	fbSetExtendedFadeTime.ipDALICommunication := ipDALICommunication;
	fbSetFadeRate.ipDALICommunication := ipDALICommunication;
	fbSetFadeTime.ipDALICommunication := ipDALICommunication;
{endregion}
5:
{region "Start Qiescent Mode"}
	fb103StartQuiescentMode(bStart := TRUE,
							eAddressType := Tc3_DALI.E_DALIAddressType.Broadcast,
							eCommandPriority := Tc3_DALI.E_DALICommandPriority.Middle);
	IF (NOT fb103StartQuiescentMode.bBusy) THEN
		fb103StartQuiescentMode(bStart:= FALSE);
		nStep := 10;
	END_IF
{endregion}
10:
{region "Query Fade Time and Fade Rate"}
	fbQueryFadeTimeFadeRate(bStart := TRUE,
							nAddress := nAddress,
							eAddressType := eAddressType,
							eCommandPriority := E_DALICommandPriority.Middle,
							eFadeTime => eFadeTime,
							eFadeRate => eFadeRate);
	IF (NOT fbQueryFadeTimeFadeRate.bBusy) THEN
		fbQueryFadeTimeFadeRate(bStart := FALSE);
		IF (eFadeTime = 0) THEN 
			bNoFadeTime := FALSE; // Check whether Fade Time is available
			nStep := 20;
		ELSE 	 
			bNoFadeTime := TRUE;
			nStep := 0;
		END_IF
	END_IF
{endregion}
20:
{region "Query Extended Fade Time"}
	fbQueryExtendedFadeTime(bStart := TRUE,
							nAddress := nAddress,
							eAddressType := eAddressType,
							eCommandPriority := E_DALICommandPriority.Middle,
							eExtendedFadeTimeBase => eExtendedFadeTimeBase,
							eExtendedFadeTimeMultiplier => eExtendedFadeTimeMultiplier);
	IF (NOT fbQueryExtendedFadeTime.bBusy) THEN
		fbQueryExtendedFadeTime(bStart := FALSE);
		nStep := 25;
		IF (eExtendedFadeTimeMultiplier = E_DALIExtendedFadeTimeMultiplier.Disabled) THEN
			eExtendedFadeTime := E_DALIExtendedFadeTime.NoFade;
		END_IF
		IF (eExtendedFadeTimeMultiplier = E_DALIExtendedFadeTimeMultiplier.Multiplier100ms) THEN
			CASE eExtendedFadeTimeBase OF
				E_DALIExtendedFadeTimeBase.Base01:	eExtendedFadeTime := E_DALIExtendedFadeTime.onehundred;
				E_DALIExtendedFadeTimeBase.Base02:	eExtendedFadeTime := E_DALIExtendedFadeTime.twohundred;
				E_DALIExtendedFadeTimeBase.Base03:	eExtendedFadeTime := E_DALIExtendedFadeTime.threehundred;
				E_DALIExtendedFadeTimeBase.Base04:	eExtendedFadeTime := E_DALIExtendedFadeTime.fourhundred;
				E_DALIExtendedFadeTimeBase.Base05:	eExtendedFadeTime := E_DALIExtendedFadeTime.fivehundred;
				E_DALIExtendedFadeTimeBase.Base06:	eExtendedFadeTime := E_DALIExtendedFadeTime.sixhundred;
				E_DALIExtendedFadeTimeBase.Base07:	eExtendedFadeTime := E_DALIExtendedFadeTime.sevenhundred;
				E_DALIExtendedFadeTimeBase.Base08:	eExtendedFadeTime := E_DALIExtendedFadeTime.eighthundred;
				E_DALIExtendedFadeTimeBase.Base09:	eExtendedFadeTime := E_DALIExtendedFadeTime.ninehundred;
				E_DALIExtendedFadeTimeBase.Base10:	eExtendedFadeTime := E_DALIExtendedFadeTime.onethousand;
				E_DALIExtendedFadeTimeBase.Base11:	eExtendedFadeTime := E_DALIExtendedFadeTime.onethousandonehundred;
				E_DALIExtendedFadeTimeBase.Base12:	eExtendedFadeTime := E_DALIExtendedFadeTime.onethousandtwohundred;
				E_DALIExtendedFadeTimeBase.Base13:	eExtendedFadeTime := E_DALIExtendedFadeTime.onethousandthreehundred;
				E_DALIExtendedFadeTimeBase.Base14:	eExtendedFadeTime := E_DALIExtendedFadeTime.onethousandfourhundred;
				E_DALIExtendedFadeTimeBase.Base15:	eExtendedFadeTime := E_DALIExtendedFadeTime.onethousandfivehundred;
				E_DALIExtendedFadeTimeBase.Base16:	eExtendedFadeTime := E_DALIExtendedFadeTime.onethousandsixhundred;
			END_CASE
		END_IF
	 	IF (eExtendedFadeTimeMultiplier = E_DALIExtendedFadeTimeMultiplier.Multiplier1s) THEN
			CASE eExtendedFadeTimeBase OF
				E_DALIExtendedFadeTimeBase.Base01:	eExtendedFadeTime := E_DALIExtendedFadeTime.onesecond;
				E_DALIExtendedFadeTimeBase.Base02:	eExtendedFadeTime := E_DALIExtendedFadeTime.twoseconds;
				E_DALIExtendedFadeTimeBase.Base03:	eExtendedFadeTime := E_DALIExtendedFadeTime.threeseconds;
				E_DALIExtendedFadeTimeBase.Base04:	eExtendedFadeTime := E_DALIExtendedFadeTime.fourseconds;
				E_DALIExtendedFadeTimeBase.Base05:	eExtendedFadeTime := E_DALIExtendedFadeTime.fiveseconds;
				E_DALIExtendedFadeTimeBase.Base06:	eExtendedFadeTime := E_DALIExtendedFadeTime.sixseconds;
				E_DALIExtendedFadeTimeBase.Base07:	eExtendedFadeTime := E_DALIExtendedFadeTime.sevenseconds;
				E_DALIExtendedFadeTimeBase.Base08:	eExtendedFadeTime := E_DALIExtendedFadeTime.eightseconds;
				E_DALIExtendedFadeTimeBase.Base09:	eExtendedFadeTime := E_DALIExtendedFadeTime.nineseconds;
				E_DALIExtendedFadeTimeBase.Base10:	eExtendedFadeTime := E_DALIExtendedFadeTime.tenseconds;
				E_DALIExtendedFadeTimeBase.Base11:	eExtendedFadeTime := E_DALIExtendedFadeTime.elevenseconds;
				E_DALIExtendedFadeTimeBase.Base12:	eExtendedFadeTime := E_DALIExtendedFadeTime.twelveseconds;
				E_DALIExtendedFadeTimeBase.Base13:	eExtendedFadeTime := E_DALIExtendedFadeTime.thirteenseconds;
				E_DALIExtendedFadeTimeBase.Base14:	eExtendedFadeTime := E_DALIExtendedFadeTime.fourteenseconds;
				E_DALIExtendedFadeTimeBase.Base15:	eExtendedFadeTime := E_DALIExtendedFadeTime.fifteenseconds;
				E_DALIExtendedFadeTimeBase.Base16:	eExtendedFadeTime := E_DALIExtendedFadeTime.sixteenseconds;
			END_CASE
		END_IF
		IF (eExtendedFadeTimeMultiplier = E_DALIExtendedFadeTimeMultiplier.Multiplier10s) THEN
			CASE eExtendedFadeTimeBase OF
				E_DALIExtendedFadeTimeBase.Base01:	eExtendedFadeTime := E_DALIExtendedFadeTime.ten1seconds;
				E_DALIExtendedFadeTimeBase.Base02:	eExtendedFadeTime := E_DALIExtendedFadeTime.twentyseconds;
				E_DALIExtendedFadeTimeBase.Base03:	eExtendedFadeTime := E_DALIExtendedFadeTime.thirtyseconds;
				E_DALIExtendedFadeTimeBase.Base04:	eExtendedFadeTime := E_DALIExtendedFadeTime.fourtyseconds;
				E_DALIExtendedFadeTimeBase.Base05:	eExtendedFadeTime := E_DALIExtendedFadeTime.fiftyseconds;
				E_DALIExtendedFadeTimeBase.Base06:	eExtendedFadeTime := E_DALIExtendedFadeTime.sixtyseconds;
				E_DALIExtendedFadeTimeBase.Base07:	eExtendedFadeTime := E_DALIExtendedFadeTime.seventyseconds;
				E_DALIExtendedFadeTimeBase.Base08:	eExtendedFadeTime := E_DALIExtendedFadeTime.eightyseconds;
				E_DALIExtendedFadeTimeBase.Base09:	eExtendedFadeTime := E_DALIExtendedFadeTime.ninetyseconds;
				E_DALIExtendedFadeTimeBase.Base10:	eExtendedFadeTime := E_DALIExtendedFadeTime.onehundredseconds;
				E_DALIExtendedFadeTimeBase.Base11:	eExtendedFadeTime := E_DALIExtendedFadeTime.onehundredtenseconds;
				E_DALIExtendedFadeTimeBase.Base12:	eExtendedFadeTime := E_DALIExtendedFadeTime.onehundredtwentyseconds;
				E_DALIExtendedFadeTimeBase.Base13:	eExtendedFadeTime := E_DALIExtendedFadeTime.onehundredthirtyseconds;
				E_DALIExtendedFadeTimeBase.Base14:	eExtendedFadeTime := E_DALIExtendedFadeTime.onehundredfourtyseconds;
				E_DALIExtendedFadeTimeBase.Base15:	eExtendedFadeTime := E_DALIExtendedFadeTime.onehundredfiftyseconds;
				E_DALIExtendedFadeTimeBase.Base16:	eExtendedFadeTime := E_DALIExtendedFadeTime.onehundredsixtyseconds;
			END_CASE
		END_IF
		IF (eExtendedFadeTimeMultiplier = E_DALIExtendedFadeTimeMultiplier.Multiplier1min) THEN
			CASE eExtendedFadeTimeBase OF
				E_DALIExtendedFadeTimeBase.Base01:	eExtendedFadeTime := E_DALIExtendedFadeTime.oneminute;
				E_DALIExtendedFadeTimeBase.Base02:	eExtendedFadeTime := E_DALIExtendedFadeTime.twominutes;
				E_DALIExtendedFadeTimeBase.Base03:	eExtendedFadeTime := E_DALIExtendedFadeTime.threeminutes;
				E_DALIExtendedFadeTimeBase.Base04:	eExtendedFadeTime := E_DALIExtendedFadeTime.fourminutes;
				E_DALIExtendedFadeTimeBase.Base05:	eExtendedFadeTime := E_DALIExtendedFadeTime.fiveminutes;
				E_DALIExtendedFadeTimeBase.Base06:	eExtendedFadeTime := E_DALIExtendedFadeTime.sixminutes;
				E_DALIExtendedFadeTimeBase.Base07:	eExtendedFadeTime := E_DALIExtendedFadeTime.sevenminutes;
				E_DALIExtendedFadeTimeBase.Base08:	eExtendedFadeTime := E_DALIExtendedFadeTime.eightminutes;
				E_DALIExtendedFadeTimeBase.Base09:	eExtendedFadeTime := E_DALIExtendedFadeTime.nineminutes;
				E_DALIExtendedFadeTimeBase.Base10:	eExtendedFadeTime := E_DALIExtendedFadeTime.tenminutes;
				E_DALIExtendedFadeTimeBase.Base11:	eExtendedFadeTime := E_DALIExtendedFadeTime.elevenminutes;
				E_DALIExtendedFadeTimeBase.Base12:	eExtendedFadeTime := E_DALIExtendedFadeTime.twelveminutes;
				E_DALIExtendedFadeTimeBase.Base13:	eExtendedFadeTime := E_DALIExtendedFadeTime.thirteenminutes;
				E_DALIExtendedFadeTimeBase.Base14:	eExtendedFadeTime := E_DALIExtendedFadeTime.fourteenminutes;
				E_DALIExtendedFadeTimeBase.Base15:	eExtendedFadeTime := E_DALIExtendedFadeTime.fifteenminutes;
				E_DALIExtendedFadeTimeBase.Base16:	eExtendedFadeTime := E_DALIExtendedFadeTime.sixteenminutes;
			END_CASE
		END_IF
	ELSE
		eExtendedFadeTime := E_DALIExtendedFadeTime.unknown;
	END_IF
{endregion}
25:
{region "Stop Qiescent Mode"}
	fb103StopQuiescentMode(	bStart := TRUE,
							eAddressType := Tc3_DALI.E_DALIAddressType.Broadcast,
							eCommandPriority := Tc3_DALI.E_DALICommandPriority.Middle);
	IF (NOT fb103StopQuiescentMode.bBusy) THEN
		fb103StopQuiescentMode(	bStart:= FALSE);
		nStep := 0;
	END_IF
{endregion}	
1000:
{region "Set Fade Time"}
	fbSetFadeTime(	bStart := TRUE,
					nAddress := nAddress,
					eAddressType := eAddressType,
					eCommandPriority := E_DALICommandPriority.Middle,
					eFadeTime := eFadeTime);
	IF (NOT fbSetFadeTime.bBusy) THEN
		fbSetFadeTime(bStart := FALSE);
		{region " Display whether Fade Time is available²}
		IF (eFadeTime = 0) THEN
			bNoFadeTime := FALSE;
		ELSE
			bNoFadeTime := TRUE;
		END_IF
		{endregion}
		nStep := 0;
	END_IF
{endregion}
1010:
{region "Set Fade Rate"}
	fbSetFadeRate(	bStart := TRUE,
					nAddress := nAddress,
					eAddressType := eAddressType,
					eCommandPriority := E_DALICommandPriority.Middle,
					eFadeRate := eFadeRate);
	IF (NOT fbSetFadeRate.bBusy) THEN
		fbSetFadeRate(bStart := FALSE);
		nStep := 0;
	END_IF
{endregion}
1020:
{region "Set Extended Fade Time"}
	CASE eExtendedFadeTime OF
		E_DALIExtendedFadeTime.NoFade:					eExtendedFadeTimeBase := E_DALIExtendedFadeTimeBase.Unknown;
														eExtendedFadeTimeMultiplier := E_DALIExtendedFadeTimeMultiplier.Disabled;
		E_DALIExtendedFadeTime.onehundred:				eExtendedFadeTimeBase := E_DALIExtendedFadeTimeBase.Base01;
														eExtendedFadeTimeMultiplier := E_DALIExtendedFadeTimeMultiplier.Multiplier100ms;
		E_DALIExtendedFadeTime.twohundred:				eExtendedFadeTimeBase := E_DALIExtendedFadeTimeBase.Base02;
														eExtendedFadeTimeMultiplier := E_DALIExtendedFadeTimeMultiplier.Multiplier100ms;
		E_DALIExtendedFadeTime.threehundred:			eExtendedFadeTimeBase := E_DALIExtendedFadeTimeBase.Base03;
														eExtendedFadeTimeMultiplier := E_DALIExtendedFadeTimeMultiplier.Multiplier100ms;
		E_DALIExtendedFadeTime.fourhundred:				eExtendedFadeTimeBase := E_DALIExtendedFadeTimeBase.Base04;
														eExtendedFadeTimeMultiplier := E_DALIExtendedFadeTimeMultiplier.Multiplier100ms;
		E_DALIExtendedFadeTime.fivehundred:				eExtendedFadeTimeBase := E_DALIExtendedFadeTimeBase.Base05;
														eExtendedFadeTimeMultiplier := E_DALIExtendedFadeTimeMultiplier.Multiplier100ms;
		E_DALIExtendedFadeTime.sixhundred:				eExtendedFadeTimeBase := E_DALIExtendedFadeTimeBase.Base06;
														eExtendedFadeTimeMultiplier := E_DALIExtendedFadeTimeMultiplier.Multiplier100ms;
		E_DALIExtendedFadeTime.sevenhundred:			eExtendedFadeTimeBase := E_DALIExtendedFadeTimeBase.Base07;
														eExtendedFadeTimeMultiplier := E_DALIExtendedFadeTimeMultiplier.Multiplier100ms;
		E_DALIExtendedFadeTime.eighthundred:			eExtendedFadeTimeBase := E_DALIExtendedFadeTimeBase.Base08;
														eExtendedFadeTimeMultiplier := E_DALIExtendedFadeTimeMultiplier.Multiplier100ms;
		E_DALIExtendedFadeTime.ninehundred:				eExtendedFadeTimeBase := E_DALIExtendedFadeTimeBase.Base09;
														eExtendedFadeTimeMultiplier := E_DALIExtendedFadeTimeMultiplier.Multiplier100ms;
		E_DALIExtendedFadeTime.onethousand:				eExtendedFadeTimeBase := E_DALIExtendedFadeTimeBase.Base10;
														eExtendedFadeTimeMultiplier := E_DALIExtendedFadeTimeMultiplier.Multiplier100ms;
		E_DALIExtendedFadeTime.onethousandonehundred:	eExtendedFadeTimeBase := E_DALIExtendedFadeTimeBase.Base11;
														eExtendedFadeTimeMultiplier := E_DALIExtendedFadeTimeMultiplier.Multiplier100ms;
		E_DALIExtendedFadeTime.onethousandtwohundred:	eExtendedFadeTimeBase := E_DALIExtendedFadeTimeBase.Base12;
														eExtendedFadeTimeMultiplier := E_DALIExtendedFadeTimeMultiplier.Multiplier100ms;
		E_DALIExtendedFadeTime.onethousandthreehundred:	eExtendedFadeTimeBase := E_DALIExtendedFadeTimeBase.Base13;
														eExtendedFadeTimeMultiplier := E_DALIExtendedFadeTimeMultiplier.Multiplier100ms;
		E_DALIExtendedFadeTime.onethousandfourhundred:	eExtendedFadeTimeBase := E_DALIExtendedFadeTimeBase.Base14;
														eExtendedFadeTimeMultiplier := E_DALIExtendedFadeTimeMultiplier.Multiplier100ms;
		E_DALIExtendedFadeTime.onethousandfivehundred:	eExtendedFadeTimeBase := E_DALIExtendedFadeTimeBase.Base15;
														eExtendedFadeTimeMultiplier := E_DALIExtendedFadeTimeMultiplier.Multiplier100ms;
		E_DALIExtendedFadeTime.onethousandsixhundred:	eExtendedFadeTimeBase := E_DALIExtendedFadeTimeBase.Base16;
														eExtendedFadeTimeMultiplier := E_DALIExtendedFadeTimeMultiplier.Multiplier100ms;
		E_DALIExtendedFadeTime.onesecond:				eExtendedFadeTimeBase := E_DALIExtendedFadeTimeBase.Base01;
														eExtendedFadeTimeMultiplier := E_DALIExtendedFadeTimeMultiplier.Multiplier1s;
		E_DALIExtendedFadeTime.twoseconds:				eExtendedFadeTimeBase := E_DALIExtendedFadeTimeBase.Base02;
														eExtendedFadeTimeMultiplier := E_DALIExtendedFadeTimeMultiplier.Multiplier1s;
		E_DALIExtendedFadeTime.threeseconds:			eExtendedFadeTimeBase := E_DALIExtendedFadeTimeBase.Base03;
														eExtendedFadeTimeMultiplier := E_DALIExtendedFadeTimeMultiplier.Multiplier1s;
		E_DALIExtendedFadeTime.fourseconds:				eExtendedFadeTimeBase := E_DALIExtendedFadeTimeBase.Base04;
														eExtendedFadeTimeMultiplier := E_DALIExtendedFadeTimeMultiplier.Multiplier1s;
		E_DALIExtendedFadeTime.fiveseconds:				eExtendedFadeTimeBase := E_DALIExtendedFadeTimeBase.Base05;
														eExtendedFadeTimeMultiplier := E_DALIExtendedFadeTimeMultiplier.Multiplier1s;
		E_DALIExtendedFadeTime.sixseconds:				eExtendedFadeTimeBase := E_DALIExtendedFadeTimeBase.Base06;
														eExtendedFadeTimeMultiplier := E_DALIExtendedFadeTimeMultiplier.Multiplier1s;
		E_DALIExtendedFadeTime.sevenseconds:			eExtendedFadeTimeBase := E_DALIExtendedFadeTimeBase.Base07;
														eExtendedFadeTimeMultiplier := E_DALIExtendedFadeTimeMultiplier.Multiplier1s;
		E_DALIExtendedFadeTime.eightseconds:			eExtendedFadeTimeBase := E_DALIExtendedFadeTimeBase.Base08;
														eExtendedFadeTimeMultiplier := E_DALIExtendedFadeTimeMultiplier.Multiplier1s;
		E_DALIExtendedFadeTime.nineseconds:				eExtendedFadeTimeBase := E_DALIExtendedFadeTimeBase.Base09;
														eExtendedFadeTimeMultiplier := E_DALIExtendedFadeTimeMultiplier.Multiplier1s;
		E_DALIExtendedFadeTime.tenseconds:				eExtendedFadeTimeBase := E_DALIExtendedFadeTimeBase.Base10;
														eExtendedFadeTimeMultiplier := E_DALIExtendedFadeTimeMultiplier.Multiplier1s;
		E_DALIExtendedFadeTime.elevenseconds:			eExtendedFadeTimeBase := E_DALIExtendedFadeTimeBase.Base11;
														eExtendedFadeTimeMultiplier := E_DALIExtendedFadeTimeMultiplier.Multiplier1s;
		E_DALIExtendedFadeTime.twelveseconds:			eExtendedFadeTimeBase := E_DALIExtendedFadeTimeBase.Base12;
														eExtendedFadeTimeMultiplier := E_DALIExtendedFadeTimeMultiplier.Multiplier1s;
		E_DALIExtendedFadeTime.thirteenseconds:			eExtendedFadeTimeBase := E_DALIExtendedFadeTimeBase.Base13;
														eExtendedFadeTimeMultiplier := E_DALIExtendedFadeTimeMultiplier.Multiplier1s;
		E_DALIExtendedFadeTime.fourteenseconds:			eExtendedFadeTimeBase := E_DALIExtendedFadeTimeBase.Base14;
														eExtendedFadeTimeMultiplier := E_DALIExtendedFadeTimeMultiplier.Multiplier1s;
		E_DALIExtendedFadeTime.fifteenseconds:			eExtendedFadeTimeBase := E_DALIExtendedFadeTimeBase.Base15;
														eExtendedFadeTimeMultiplier := E_DALIExtendedFadeTimeMultiplier.Multiplier1s;
		E_DALIExtendedFadeTime.sixteenseconds:			eExtendedFadeTimeBase := E_DALIExtendedFadeTimeBase.Base16;
														eExtendedFadeTimeMultiplier := E_DALIExtendedFadeTimeMultiplier.Multiplier1s;
		E_DALIExtendedFadeTime.ten1seconds:				eExtendedFadeTimeBase := E_DALIExtendedFadeTimeBase.Base01;
														eExtendedFadeTimeMultiplier := E_DALIExtendedFadeTimeMultiplier.Multiplier10s;
		E_DALIExtendedFadeTime.twentyseconds:			eExtendedFadeTimeBase := E_DALIExtendedFadeTimeBase.Base02;
														eExtendedFadeTimeMultiplier := E_DALIExtendedFadeTimeMultiplier.Multiplier10s;
		E_DALIExtendedFadeTime.thirtyseconds:			eExtendedFadeTimeBase := E_DALIExtendedFadeTimeBase.Base03;
														eExtendedFadeTimeMultiplier := E_DALIExtendedFadeTimeMultiplier.Multiplier10s;
		E_DALIExtendedFadeTime.fourtyseconds:			eExtendedFadeTimeBase := E_DALIExtendedFadeTimeBase.Base04;
														eExtendedFadeTimeMultiplier := E_DALIExtendedFadeTimeMultiplier.Multiplier10s;
		E_DALIExtendedFadeTime.fiftyseconds:			eExtendedFadeTimeBase := E_DALIExtendedFadeTimeBase.Base05;
														eExtendedFadeTimeMultiplier := E_DALIExtendedFadeTimeMultiplier.Multiplier10s;
		E_DALIExtendedFadeTime.sixtyseconds:			eExtendedFadeTimeBase := E_DALIExtendedFadeTimeBase.Base06;
														eExtendedFadeTimeMultiplier := E_DALIExtendedFadeTimeMultiplier.Multiplier10s;
		E_DALIExtendedFadeTime.seventyseconds:			eExtendedFadeTimeBase := E_DALIExtendedFadeTimeBase.Base07;
														eExtendedFadeTimeMultiplier := E_DALIExtendedFadeTimeMultiplier.Multiplier10s;
		E_DALIExtendedFadeTime.eightyseconds:			eExtendedFadeTimeBase := E_DALIExtendedFadeTimeBase.Base08;
														eExtendedFadeTimeMultiplier := E_DALIExtendedFadeTimeMultiplier.Multiplier10s;
		E_DALIExtendedFadeTime.ninetyseconds:			eExtendedFadeTimeBase := E_DALIExtendedFadeTimeBase.Base09;
														eExtendedFadeTimeMultiplier := E_DALIExtendedFadeTimeMultiplier.Multiplier10s;
		E_DALIExtendedFadeTime.onehundredseconds:		eExtendedFadeTimeBase := E_DALIExtendedFadeTimeBase.Base10;
														eExtendedFadeTimeMultiplier := E_DALIExtendedFadeTimeMultiplier.Multiplier10s;
		E_DALIExtendedFadeTime.onehundredtenseconds:	eExtendedFadeTimeBase := E_DALIExtendedFadeTimeBase.Base11;
														eExtendedFadeTimeMultiplier := E_DALIExtendedFadeTimeMultiplier.Multiplier10s;
		E_DALIExtendedFadeTime.onehundredtwentyseconds:	eExtendedFadeTimeBase := E_DALIExtendedFadeTimeBase.Base12;
														eExtendedFadeTimeMultiplier := E_DALIExtendedFadeTimeMultiplier.Multiplier10s;
		E_DALIExtendedFadeTime.onehundredthirtyseconds:	eExtendedFadeTimeBase := E_DALIExtendedFadeTimeBase.Base13;
														eExtendedFadeTimeMultiplier := E_DALIExtendedFadeTimeMultiplier.Multiplier10s;
		E_DALIExtendedFadeTime.onehundredfourtyseconds:	eExtendedFadeTimeBase := E_DALIExtendedFadeTimeBase.Base14;
														eExtendedFadeTimeMultiplier := E_DALIExtendedFadeTimeMultiplier.Multiplier10s;
		E_DALIExtendedFadeTime.onehundredfiftyseconds:	eExtendedFadeTimeBase := E_DALIExtendedFadeTimeBase.Base15;
														eExtendedFadeTimeMultiplier := E_DALIExtendedFadeTimeMultiplier.Multiplier10s;
		E_DALIExtendedFadeTime.onehundredsixtyseconds:	eExtendedFadeTimeBase := E_DALIExtendedFadeTimeBase.Base16;
														eExtendedFadeTimeMultiplier := E_DALIExtendedFadeTimeMultiplier.Multiplier10s;
		E_DALIExtendedFadeTime.oneminute:				eExtendedFadeTimeBase := E_DALIExtendedFadeTimeBase.Base01;
														eExtendedFadeTimeMultiplier := E_DALIExtendedFadeTimeMultiplier.Multiplier1min;
		E_DALIExtendedFadeTime.twominutes:				eExtendedFadeTimeBase := E_DALIExtendedFadeTimeBase.Base02;
														eExtendedFadeTimeMultiplier := E_DALIExtendedFadeTimeMultiplier.Multiplier1min;
		E_DALIExtendedFadeTime.threeminutes:			eExtendedFadeTimeBase := E_DALIExtendedFadeTimeBase.Base03;
														eExtendedFadeTimeMultiplier := E_DALIExtendedFadeTimeMultiplier.Multiplier1min;
		E_DALIExtendedFadeTime.fourminutes:				eExtendedFadeTimeBase := E_DALIExtendedFadeTimeBase.Base04;
														eExtendedFadeTimeMultiplier := E_DALIExtendedFadeTimeMultiplier.Multiplier1min;
		E_DALIExtendedFadeTime.fiveminutes:				eExtendedFadeTimeBase := E_DALIExtendedFadeTimeBase.Base05;
														eExtendedFadeTimeMultiplier := E_DALIExtendedFadeTimeMultiplier.Multiplier1min;
		E_DALIExtendedFadeTime.sixminutes:				eExtendedFadeTimeBase := E_DALIExtendedFadeTimeBase.Base06;
														eExtendedFadeTimeMultiplier := E_DALIExtendedFadeTimeMultiplier.Multiplier1min;
		E_DALIExtendedFadeTime.sevenminutes:			eExtendedFadeTimeBase := E_DALIExtendedFadeTimeBase.Base07;
														eExtendedFadeTimeMultiplier := E_DALIExtendedFadeTimeMultiplier.Multiplier1min;
		E_DALIExtendedFadeTime.eightminutes:			eExtendedFadeTimeBase := E_DALIExtendedFadeTimeBase.Base08;
														eExtendedFadeTimeMultiplier := E_DALIExtendedFadeTimeMultiplier.Multiplier1min;
		E_DALIExtendedFadeTime.nineminutes:				eExtendedFadeTimeBase := E_DALIExtendedFadeTimeBase.Base09;
														eExtendedFadeTimeMultiplier := E_DALIExtendedFadeTimeMultiplier.Multiplier1min;
		E_DALIExtendedFadeTime.tenminutes:				eExtendedFadeTimeBase := E_DALIExtendedFadeTimeBase.Base10;
														eExtendedFadeTimeMultiplier := E_DALIExtendedFadeTimeMultiplier.Multiplier1min;
		E_DALIExtendedFadeTime.elevenminutes:			eExtendedFadeTimeBase := E_DALIExtendedFadeTimeBase.Base11;
														eExtendedFadeTimeMultiplier := E_DALIExtendedFadeTimeMultiplier.Multiplier1min;
		E_DALIExtendedFadeTime.twelveminutes:			eExtendedFadeTimeBase := E_DALIExtendedFadeTimeBase.Base12;
														eExtendedFadeTimeMultiplier := E_DALIExtendedFadeTimeMultiplier.Multiplier1min;
		E_DALIExtendedFadeTime.thirteenminutes:			eExtendedFadeTimeBase := E_DALIExtendedFadeTimeBase.Base13;
														eExtendedFadeTimeMultiplier := E_DALIExtendedFadeTimeMultiplier.Multiplier1min;
		E_DALIExtendedFadeTime.fourteenminutes:			eExtendedFadeTimeBase := E_DALIExtendedFadeTimeBase.Base14;
														eExtendedFadeTimeMultiplier := E_DALIExtendedFadeTimeMultiplier.Multiplier1min;
		E_DALIExtendedFadeTime.fifteenminutes:			eExtendedFadeTimeBase := E_DALIExtendedFadeTimeBase.Base15;
														eExtendedFadeTimeMultiplier := E_DALIExtendedFadeTimeMultiplier.Multiplier1min;
		E_DALIExtendedFadeTime.sixteenminutes:			eExtendedFadeTimeBase := E_DALIExtendedFadeTimeBase.Base16;
														eExtendedFadeTimeMultiplier := E_DALIExtendedFadeTimeMultiplier.Multiplier1min;
		E_DALIExtendedFadeTime.unknown:					eExtendedFadeTimeBase := E_DALIExtendedFadeTimeBase.Unknown;
														eExtendedFadeTimeMultiplier := E_DALIExtendedFadeTimeMultiplier.Unknown;
	END_CASE
	fbSetExtendedFadeTime(	bStart := TRUE,
							nAddress := nAddress,
							eAddressType := eAddressType,
							eCommandPriority := E_DALICommandPriority.Middle,
							eExtendedFadeTimeBase := eExtendedFadeTimeBase,
							eExtendedFadeTimeMultiplier := eExtendedFadeTimeMultiplier);
	IF (NOT fbSetExtendedFadeTime.bBusy) THEN
		fbSetExtendedFadeTime(bStart := FALSE);
		nStep := 0;
	END_IF
{endregion}
END_CASE

END_FUNCTION_BLOCK

// ---- POUs/DALI/DALI_Setup/FBs/FB_Part103Addressing.TcPOU
FUNCTION_BLOCK FB_Part103Addressing
VAR_INPUT
	ipDALICommunication			:	I_DALICommunication;
END_VAR
VAR_OUTPUT
	bBusy						:	BOOL;
END_VAR
VAR
	{region "Visu"}
	bScanDevices				:	BOOL;
	bStartChangeAddress			:	BOOL;
	bStartRandomAddressing		:	BOOL;
	nStartAddress				:	BYTE;
	bNewInstallation			:	BOOL;
	bOpticalFeedback			:	BOOL;
	bHideWaitSymbol				:	BOOL := TRUE;
	{endregion}
	nStep						:	INT;
	nAddress					:	INT;
	aChangeAddressList			:	ARRAY [0..63] OF ST_DALIChangeAddressList;
	aShortAddress				:	ARRAY [0..63] OF INT;
	aNoShortAddress				:	ARRAY [0..63] OF BOOL;
	nRow						:	INT;
	nHideLine					:	INT; // Variable to find out how many rows are used

	fb103StartQuiescentMode		:	FB_DALI103StartQuiescentMode(0);
	fb103StopQuiescentMode		:	FB_DALI103StopQuiescentMode(0);
	fb103Addressing				:	FB_DALI103Addressing(0);
	fb103QueryRandomAddress		:	FB_DALI103QueryRandomAddress(0);
	fb103ChangeAddresses		:	FB_DALI103ChangeAddresses(0);
END_VAR

{region "Detect Commands"}
IF (bStartRandomAddressing AND (nStep = 0)) THEN
	nStep := 5;
	bStartRandomAddressing := FALSE;
	bHideWaitSymbol := FALSE;
END_IF

IF (bScanDevices AND (nStep = 0)) THEN
	nStep := 20;
	nAddress :=0;
	bScanDevices := FALSE;
	bHideWaitSymbol := FALSE;
END_IF

IF (bStartChangeAddress AND (nStep = 0)) THEN
	nStep := 60;
	bStartChangeAddress := FALSE;
	bHideWaitSymbol := FALSE;
END_IF
{endregion}
{region "Manage Dialog Selection}
IF (nStep = 0) THEN
	bBusy := FALSE;
ELSE
	bBusy := TRUE;
END_IF
{endregion}	 
{region "Execute Commands"}
CASE nStep OF
0:
{region "Init"}
	bScanDevices := FALSE;
	bStartChangeAddress := FALSE;
	bStartRandomAddressing := FALSE;
	bHideWaitSymbol := TRUE;

	fb103StartQuiescentMode.ipDALICommunication := ipDALICommunication;
	fb103StopQuiescentMode.ipDALICommunication := ipDALICommunication;
	fb103Addressing.ipDALICommunication := ipDALICommunication;
	fb103QueryRandomAddress.ipDALICommunication := ipDALICommunication;
	fb103ChangeAddresses.ipDALICommunication := ipDALICommunication;
{endregion}
5:
{region "Start Qiescent Mode"}
	fb103StartQuiescentMode(bStart := TRUE,
							eAddressType := Tc3_DALI.E_DALIAddressType.Broadcast,
							eCommandPriority := Tc3_DALI.E_DALICommandPriority.Middle);
	IF (NOT fb103StartQuiescentMode.bBusy) THEN
		fb103StartQuiescentMode(bStart:= FALSE);
		nStep := 10;
	END_IF
{endregion}
10:
{region "RandomAddressing"}
	IF bNewInstallation THEN
		fb103Addressing.nOptions := Tc3_DALI.GVL.cCompleteNewInstallation;
	END_IF

	IF bOpticalFeedback THEN
		fb103Addressing.nOptions := Tc3_DALI.GVL.cOpticalFeedback;
	END_IF

	IF bNewInstallation AND bOpticalFeedback THEN
		fb103Addressing.nOptions := Tc3_DALI.GVL.cCompleteNewInstallation OR Tc3_DALI.GVL.cOpticalFeedback;
	END_IF
	fb103Addressing(bStart := TRUE,
					nStartWithShortAddress := nStartAddress);
	IF (NOT fb103Addressing.bBusy) THEN
		fb103Addressing(bStart := FALSE);
		nStep := 15;
	END_IF
{endregion}
15:
{region "Stop Qiescent Mode"}
	fb103StopQuiescentMode(	bStart := TRUE,
							eAddressType := Tc3_DALI.E_DALIAddressType.Broadcast,
							eCommandPriority := Tc3_DALI.E_DALICommandPriority.Middle);
	IF (NOT fb103StopQuiescentMode.bBusy) THEN
		fb103StopQuiescentMode(	bStart:= FALSE);
		nStep := 0;
	END_IF
{endregion}
{region "Read Existing Addresses"}
20:
{region "Start Qiescent Mode"}
	fb103StartQuiescentMode(bStart := TRUE,
							eAddressType := Tc3_DALI.E_DALIAddressType.Broadcast,
							eCommandPriority := Tc3_DALI.E_DALICommandPriority.Middle);
	IF (NOT fb103StartQuiescentMode.bBusy) THEN
		fb103StartQuiescentMode(bStart:= FALSE);
		nStep := 30;
	END_IF
{endregion}
30:
	// Query of the new random addresses to find out which short addresses are existing.
	fb103QueryRandomAddress (	bStart := TRUE,
								nAddress := TO_BYTE(nAddress),
								eAddressType := Tc3_DALI.E_DALIAddressType.Short,
								nRandomAddress => aChangeAddressList[nAddress].nRandomAddress);
	IF (NOT fb103QueryRandomAddress.bBusy) THEN
		fb103QueryRandomAddress(bStart := FALSE);
		nAddress := nAddress + 1;
		IF (nAddress > 63) THEN
			nStep := 40;
		END_IF
	END_IF
40:
	// Write the existing short addresses into the table 
	nRow := 0;
	FOR nAddress := 0 TO 63 DO
		IF (aChangeAddressList[nAddress].nRandomAddress > 0) THEN
			aChangeAddressList[nRow].nOldAddress := TO_BYTE(nAddress);
			nRow := nRow + 1;
		END_IF
	END_FOR
	nStep := 50;
50:
	// Hide unused rows in the table
	nHideLine := 0;
	FOR nAddress := 0 TO 63 DO 
		IF (aChangeAddressList[nAddress].nRandomAddress <> 0) THEN
			aShortAddress[nHideLine] := nAddress;
			nHideLine := nHideLine + 1;
		END_IF
	END_FOR
	FOR nAddress := nHideLine TO 63 DO 
		aNoShortAddress[nAddress] := TRUE;
	END_FOR
	FOR nAddress := 0 TO (nHideLine - 1) DO
		aNoShortAddress[nAddress] := FALSE;
	END_FOR
	aChangeAddressList[nHideLine].nOldAddress := 255;
	FOR nAddress := 0 TO nHideLine DO
		aChangeAddressList[nAddress].nNewAddress := aChangeAddressList[nAddress].nOldAddress;
	END_FOR
	nStep := 55;
{endregion}
55:
{region "Stop Qiescent Mode"}
	fb103StopQuiescentMode(	bStart := TRUE,
							eAddressType := Tc3_DALI.E_DALIAddressType.Broadcast,
							eCommandPriority := Tc3_DALI.E_DALICommandPriority.Middle);
	IF (NOT fb103StopQuiescentMode.bBusy) THEN
		fb103StopQuiescentMode(	bStart:= FALSE);
		nStep := 0;
	END_IF
{endregion}
60:
{region "Write Changed Addresses}
	fb103ChangeAddresses(	bStart := TRUE,
							aChangeAddressList := aChangeAddressList);
	IF (NOT fb103ChangeAddresses.bBusy) THEN
		fb103ChangeAddresses(	bStart := FALSE,
								aChangeAddressList := aChangeAddressList);
		nStep := 70;
	END_IF
{endregion}
70:
{region "Write New Address To Old Address}
	FOR nAddress := 0 TO 63 DO
		aChangeAddressList[nAddress].nOldAddress := aChangeAddressList[nAddress].nNewAddress;
	END_FOR
	nStep := 0;
{endregion}
END_CASE

END_FUNCTION_BLOCK

// ---- POUs/DALI/PRGs/EnergyData/P_DALI_Energy_Line.TcPOU
(*
EnergyReporting reads ActiveEnergy (part 252) for all present ballasts on all (configured) DALI-lines where GVL_DALI.g_arrEnergyData[*DALI-line*,*ballast*].bHasEnergyData is TRUE.
Results are stored in GVL_DALI.g_arrEnergyData[*DALI-line*,*ballast*].fActiveEnergy. Energy Data for individual ballasts is NOT persistent.
The engergy sum per DALI-Line (Wh) and Total Energy (kWh) are persistent.

If bCheckActiveEnergy is TRUE, all present ballasts are queried for ActiveEnergy and bHasEnergyData is updated accordingly.
This will result in errors for any ballast that does not comply with part 252.
Errors will not be triggered for activations where bCheckActiveEnergy is FALSE.

After shutdown or download to PLC EnergyReporting is activated automatically internally with bCheckActiveEnergy set to TRUE

EnergyReporting is activated automatically at TOD 0:00, 6:00, 12:00, 18:00 (configurable)

NB:	The priority of commands are set to "middle" internally. Updating all lines will take a couple of minutes to finish, so be patient.
	Other critical commands on the DALI-lines take priotity.
	Add appropriate communication immediately after configuration of a new KL6821 terminal.
	That is, arrfbDALI_EnergyReporting[*DALI-Line*].ipDALICommunication := P_DALI_Background.arrfbKL6821Communication[*DALI-Line*];
*)


PROGRAM P_DALI_Energy_Line
VAR
	arrfbDALI_EnergyReporting	: ARRAY[1..SH_Light.DALI_Param.MAX_DALIV2_LINES] OF FB_DALI_EnergyReporting;
	fbDALI_EnergyDataManagement	: SH_Light.FB_DALI_EnergyDataManagement;
	nNumOfEnergyLines			: BYTE;
	bReadEnergyDataAllLines		: BOOL;
	bReportingDone				: BOOL;
	fbRTrig_ReportingDone		: R_TRIG;
	bRTrigReportingDone			: BOOL;
	
	//Task scheduling
	stLocalSystemTime 		: TIMESTRUCT;
	fbLocalSystemTime 		: FB_LocalSystemTime;
	bGetTime 				: BOOL := TRUE;
	tTimeOut 				: TIME := DEFAULT_ADS_TIMEOUT;
	bLocalSystemTimeValid	: BOOL;
	tzID       				: E_TimeZoneID := eTimeZoneID_Invalid;
	
	tdSystemTime			: TOD;
	btestTodCompare			: BOOL;
	
	
END_VAR
VAR CONSTANT
	tdMidnight						: TOD := TOD#0:0:0;
	tdMorning						: TOD := TOD#6:0:0;
	tdMidDay						: TOD := TOD#12:0:0;
	tdEvening						: TOD := TOD#18:0:0;
	tCheckDuration					: TIME:= T#5S;
	tdTestsum						: TOD := (tdMidnight + tCheckDuration);
END_VAR

VAR PERSISTENT
	arrDaliLineEnergySumWh				: ARRAY[1..SH_Light.DALI_Param.MAX_DALIV2_LINES] OF LREAL;
	fTotalEnergyWh						: LREAL;
	nMaxControlGearOperatingHours		: UINT;
END_VAR


arrfbDALI_EnergyReporting[1].ipDALICommunication := P_DALI_Background.arrfbKL6821Communication[1];
arrfbDALI_EnergyReporting[2].ipDALICommunication := P_DALI_Background.arrfbKL6821Communication[2];
arrfbDALI_EnergyReporting[3].ipDALICommunication := P_DALI_Background.arrfbKL6821Communication[3];
//arrfbDALI_EnergyReporting[4].ipDALICommunication := P_DALI_Background.arrfbKL6821Communication[4];
//arrfbDALI_EnergyReporting[5].ipDALICommunication := P_DALI_Background.arrfbKL6821Communication[5];
//arrfbDALI_EnergyReporting[6].ipDALICommunication := P_DALI_Background.arrfbKL6821Communication[6]; // for more update SH_Light.DALI_Param.MAX_DALIV2_LINES

nNumOfEnergyLines := 3;

fbLocalSystemTime(
	sNetID:= '', 
	bEnable:= bGetTime, 
	dwCycle:= 2, // cycle time (in seconds) , Synchronization  every 2 seconds.
	dwOpt:= 1, //Bit 0: If this is set, the Windows system time is additionally synchronized cyclically with the hardware clock (RTC) (corresponds to the function NT_SetTimeToRTCTime).
	tTimeout:= tTimeOut, 
	bValid=> bLocalSystemTimeValid, 
	systemTime=> stLocalSystemTime, 
	tzID=> tzID);
	
tdSystemTime := SYSTEMTIME_TO_TOD(systemTime := stLocalSystemTime);
IF	((tdSystemTime > tdMidnight AND tdSystemTime < (tdMidnight + tCheckDuration)) OR (tdSystemTime > tdMorning AND tdSystemTime < (tdMorning + tCheckDuration)) OR
	(tdSystemTime > tdMidDay AND tdSystemTime < (tdMidDay + tCheckDuration)) OR (tdSystemTime > tdEvening AND tdSystemTime < (tdEvening + tCheckDuration))) THEN
	bReadEnergyDataAllLines := TRUE;
END_IF

fbDALI_EnergyDataManagement(
	NumOfEnergyLines				:= nNumOfEnergyLines,
	bReadEnergyDataAllLines 		:= bReadEnergyDataAllLines,
	arrfbDALI_EnergyReporting		:= arrfbDALI_EnergyReporting,
	arrDaliLineEnergySum			:= arrDaliLineEnergySumWH,
	fTotalEnergyWh					:= fTotalEnergyWh,
	nMaxControlGearOperatingHours	:= nMaxControlGearOperatingHours,
	bReportingDone					=> bReportingDone
);
GVL_AHDataModbus.nTotalEnergy10kWh := TO_UINT(TRUNC(fTotalEnergyWh*EXPT(10,-4)));  //FB_DALI_EnergyDataManagement makes sure only positive values are returned. As so, conversion from REAL to UINT is appropriate
GVL_AHDataModbus.nMaxControlGearOperatingHours := nMaxControlGearOperatingHours;

END_PROGRAM

// ---- POUs/EnOcean/P_EnOcean.TcPOU
PROGRAM P_EnOcean
VAR
	fbKL6581			: FB_KL6581;
	stKL6581_in  AT %I* : KL6581_INPUT;
	stKL6581_out AT %Q*	: KL6581_OUTPUT;
	stKL6581			: STR_KL6581;
	bInitCom			: BOOL := TRUE;
	
	arrEnOcean_Search	: ARRAY [1..8] OF FB_EnOcean_Search;
	nSearchIdx			: BYTE;
	bSerach				: BOOL;
	arrDevices			: ARRAY [1..8] OF INT;
	arrID					: ARRAY [1..8, 0..255] OF DWORD;

	//Trykknapper Atrium
	fbAtriumNiveau_Tryk_PladeB_Old				: FB_Rec_RPS_Switch;
	fbAtriumNiveau_Tryk_PladeB						: FB_Rec_RPS_Switch;
	fbAtriumNiveau_Tryk_Sevice						: FB_Rec_RPS_Switch;

	//Trykknapper på gange
	fbGang_4_413_Tryk_Pendler    						: FB_Rec_RPS_Switch;	
	
	//Trykknapper i rum
	fbRum_3_429_Tryk_Indgang							: FB_Rec_RPS_Switch;
	fbRum_3_429_Tryk_Ekstra							: FB_Rec_RPS_Switch;
	
	fbRum_4_407_Tryk_Indgang1						: FB_Rec_RPS_Switch;
	fbRum_4_407_Tryk_Indgang2						: FB_Rec_RPS_Switch;
	
	fbRum_4_411_Tryk_Indgang							: FB_Rec_RPS_Switch;
	fbRum_4_411_Tryk_Ekstra							: FB_Rec_RPS_Switch;
	
	//fbRum_1_215_Tryk											: FB_Rec_RPS_Switch;
	
END_VAR

VAR CONSTANT
	byNode_1: BYTE := 1;
	byNode_2: BYTE := 2;
	byNode_3: BYTE := 3;
	byNode_4: BYTE := 4;
	byNode_5: BYTE := 5;
	byNode_6: BYTE := 6;
	byNode_7: BYTE := 7;
	byNode_8: BYTE := 8;
END_VAR


(* Kommunikation mit der KL6581. *)
(* Communication with the KL6581. *)
fbKL6581(
	bInit			:= bInitCom,
	nIdx			:= 2,
	stKL6581_in		:= stKL6581_In,
	stKL6581_out	:= stKL6581_Out,
	bReady			=> ,
	bBusy			=> ,
	bError			=> ,
	iErrorID		=> ,
	str_KL6581		=> stKL6581);
	
GVL_AHDataModbus.EnOceanError	:= TO_UINT(fbKL6581.iErrorID);

(* Warten bis der Kommunikationsbaustein initialisiert wurde.*)
(* Wait until the communication function block has been initialized. *)
IF (NOT fbKL6581.bReady) THEN
	RETURN;
END_IF

FOR nSearchIdx:= 1 TO 8 DO
	arrEnOcean_Search[nSearchIdx](
		bStart:= TRUE, 
		str_KL6581:= stKL6581 , 
		byNode:= nSearchIdx, 
		bReceive=> , 
		iDevices=>arrDevices[nSearchIdx] , 
		ar_ID=> );
		
		MEMCPY(ADR(arrID[nSearchIdx,0]), ADR(arrEnOcean_Search[nSearchIdx].ar_ID), SIZEOF(arrEnOcean_Search[nSearchIdx].ar_ID)); 
END_FOR

//Atrium
A_AtriumNiveau();

//Gange
A_Gang_4_413();

//Rum
A_Rum_3_429();
A_Rum_4_407();
A_Rum_4_411();

ACTION A_AtriumNiveau:
fbAtriumNiveau_Tryk_PladeB_Old(
	str_KL6581:=stKL6581 , 
	byNode:=0, 
	dw_ID:= 16#0029EE85, 
	str_EnOceanSwitch=> GVL_EnOcean.strEnOceanSwitch_AtriumNiveau_PladeB_Old,
	by_Node=> , 
	bReceive=> );
	
	fbAtriumNiveau_Tryk_PladeB(
	str_KL6581:=stKL6581 , 
	byNode:=0, 
	dw_ID:= 16#0029B92D, 
	str_EnOceanSwitch=> GVL_EnOcean.strEnOceanSwitch_AtriumNiveau_PladeB,
	by_Node=> , 
	bReceive=> );
	
(*
fbAtriumNiveau_Tryk_Sevice(
	str_KL6581:=stKL6581 , 
	byNode:=0, 
	dw_ID:= 16#00FEE4FE87, 
	str_EnOceanSwitch=> GVL_EnOcean.strEnOceanSwitch_AtriumNiveau_Service, 
	by_Node=> , 
	bReceive=> );
*)
END_ACTION

ACTION A_Gang_4_413:
fbGang_4_413_Tryk_Pendler(
	str_KL6581:=stKL6581 , 
	byNode:=byNode_2, 
	dw_ID:= 16#0029AAC6, 
	str_EnOceanSwitch=> GVL_EnOcean.strEnOceanSwitch_Gang_4_413_Pendler, 
	by_Node=> , 
	bReceive=> );
END_ACTION

ACTION A_Rum_3_429:
fbRum_3_429_Tryk_Indgang(
	str_KL6581:=stKL6581 , 
	byNode:=byNode_2, 
	dw_ID:= 16#0029AD76, 
	str_EnOceanSwitch=> GVL_EnOcean.strEnOceanSwitch_Rum_3_429_Indgang, 
	by_Node=> , 
	bReceive=> );
	
	fbRum_3_429_Tryk_Ekstra(
	str_KL6581:=stKL6581 , 
	byNode:=byNode_2, 
	dw_ID:= 16#0029ABAC, 
	str_EnOceanSwitch=> GVL_EnOcean.strEnOceanSwitch_Rum_3_429_Ekstra, 
	by_Node=> , 
	bReceive=> );
END_ACTION

ACTION A_Rum_4_407:
fbRum_4_407_Tryk_Indgang1(
	str_KL6581:=stKL6581 , 
	byNode:=byNode_2, 
	dw_ID:= 16#0, 
	str_EnOceanSwitch=> GVL_EnOcean.strEnOceanSwitch_Rum_4_407_Indgang1, 
	by_Node=> , 
	bReceive=> );
	
	fbRum_4_407_Tryk_Indgang2(
	str_KL6581:=stKL6581 , 
	byNode:=byNode_2, 
	dw_ID:= 16#0, 
	str_EnOceanSwitch=> GVL_EnOcean.strEnOceanSwitch_Rum_4_407_Indgang2, 
	by_Node=> , 
	bReceive=> );
END_ACTION

ACTION A_Rum_4_411:
fbRum_4_411_Tryk_Indgang(
	str_KL6581:=stKL6581 , 
	byNode:=byNode_2, 
	dw_ID:= 16#0029ABB2, 
	str_EnOceanSwitch=> GVL_EnOcean.strEnOceanSwitch_Rum_4_411_Indgang, 
	by_Node=> , 
	bReceive=> );
	
	fbRum_4_411_Tryk_Ekstra(
	str_KL6581:=stKL6581 , 
	byNode:=byNode_2, 
	dw_ID:= 16#0029AADD, 
	str_EnOceanSwitch=> GVL_EnOcean.strEnOceanSwitch_Rum_4_411_Ekstra, 
	by_Node=> , 
	bReceive=> );
END_ACTION

END_PROGRAM

// ---- POUs/MAIN.TcPOU
PROGRAM MAIN
VAR
	nAlive: INT;
	breset: BOOL;
	nDemoVariable : INT;
	nCX8200_State	AT %I*	: UINT;
END_VAR

VAR PERSISTENT
	nDemoVar_Persist: INT;
END_VAR

nAlive:= nAlive + 1;
GVL_AHDataModbus.nCX8200_State_MB := nCX8200_State;

//Håndterer vedvarende data
	P_SystemDK.M_nCyclic(bReset := breset );
//Håndterer DALI-diagnostik (run once)
	P_DALI_DIAG();
//Håndterer adressering		
	DALI_Commissioning();
//Håndterer energirapportering
	P_DALI_Energy_Line();
//Håndterer moodbus-kommunikation (kun PLC-oversigt)
	P_AHModbusComm();

//Håndterer individuel lyskontrol i lokaler
	//Gange
	P_Gang_3_409();
	P_Gang_4_410A();
	P_Gang_4_413();

	
	//Rum
	P_Rum_3_429();
	P_Rum_4_407();
	P_Rum_4_411();
	
//Testprogrammer
	//P_DALI_Energy_Firmware_Test();

END_PROGRAM

// ---- POUs/Alle_Rum/Gange/Gang_3_409/Visualization_4_308_1.TcVIS
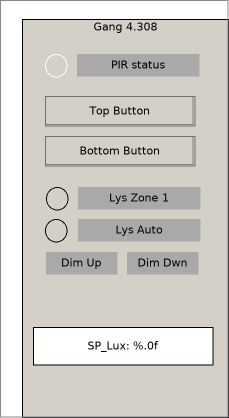
VISUALIZATION Visualization_4_308_1  // 229x418
    RoundedRectangle (22,19 207x399), "Gang 4.308"
    Rectangle (33,327 180x38), "SP_Lux: %.0f", text variable: P_Gang_4_308.arrfbLysGruppe[1].fbLightCtrl.fLuxZone1
    Button (45,96 150x30), "Top Button"
        tap P_Gang_4_308.bButtonZone1_Visu
    Button (45,136 150x30), "Bottom Button"
        tap P_Gang_4_308.bBottomButtonZone1_Visu
    Ellipse (46,187 22x23), colour toggle: P_Gang_4_308.fbLys.fbLightCtrl.bOnZone1
    Rectangle (78,187 122x22), "Lys Zone 1"
    Rectangle (46,252 71x22), "Dim Up", colour toggle: P_Gang_4_308.arrfbLysGruppe[1].fbLightCtrl.bDimUp
    Rectangle (127,252 71x22), "Dim Dwn", colour toggle: P_Gang_4_308.arrfbLysGruppe[1].fbLightCtrl.bDimDwn
    Ellipse (45,219 22x23), colour toggle: P_Gang_4_308.arrfbLysGruppe[1].fbLightCtrl.bAutoZone1
    Rectangle (78,219 122x22), "Lys Auto"
    Ellipse (45,54 22x23), colour toggle: P_Gang_4_308.arrfbLysGruppe[1].fbLightCtrl.bPIR
    Rectangle (77,54 122x22), "PIR status"
END_VISUALIZATION

// ---- POUs/Alle_Rum/Gange/Gang_4_313/Visualization_4_308_1_1.TcVIS
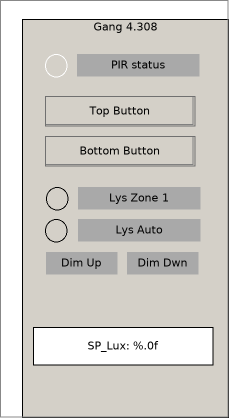
VISUALIZATION Visualization_4_308_1_1  // 229x418
    RoundedRectangle (22,19 207x399), "Gang 4.308"
    Rectangle (33,327 180x38), "SP_Lux: %.0f", text variable: P_Gang_4_308.arrfbLysGruppe[1].fbLightCtrl.fLuxZone1
    Button (45,96 150x30), "Top Button"
        tap P_Gang_4_308.bButtonZone1_Visu
    Button (45,136 150x30), "Bottom Button"
        tap P_Gang_4_308.bBottomButtonZone1_Visu
    Ellipse (46,187 22x23), colour toggle: P_Gang_4_308.fbLys.fbLightCtrl.bOnZone1
    Rectangle (78,187 122x22), "Lys Zone 1"
    Rectangle (46,252 71x22), "Dim Up", colour toggle: P_Gang_4_308.arrfbLysGruppe[1].fbLightCtrl.bDimUp
    Rectangle (127,252 71x22), "Dim Dwn", colour toggle: P_Gang_4_308.arrfbLysGruppe[1].fbLightCtrl.bDimDwn
    Ellipse (45,219 22x23), colour toggle: P_Gang_4_308.arrfbLysGruppe[1].fbLightCtrl.bAutoZone1
    Rectangle (78,219 122x22), "Lys Auto"
    Ellipse (45,54 22x23), colour toggle: P_Gang_4_308.arrfbLysGruppe[1].fbLightCtrl.bPIR
    Rectangle (77,54 122x22), "PIR status"
END_VISUALIZATION

// ---- POUs/Alle_Rum/Rum_Med_DALI_Pir/Rum_4_411/Visualization_5_356_2_1_1_3_2.TcVIS
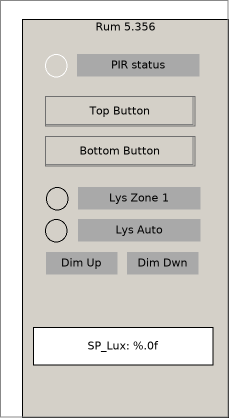
VISUALIZATION Visualization_5_356_2_1_1_3_2  // 229x418
    RoundedRectangle (22,19 207x399), "Rum 5.356"
    Rectangle (33,327 180x38), "SP_Lux: %.0f", text variable: P_Rum_5_356.arrfbLysGruppe[1].fbLightCtrl.fLuxZone1
    Button (45,96 150x30), "Top Button"
        tap P_Rum_5_356.bTopButtonZone1_Visu
    Button (45,136 150x30), "Bottom Button"
        tap P_Rum_5_356.bBottomButtonZone1_Visu
    Ellipse (46,187 22x23), colour toggle: P_Rum_5_356.arrfbLysGruppe[1].fbLightCtrl.bOnZone1
    Rectangle (78,187 122x22), "Lys Zone 1"
    Rectangle (46,252 71x22), "Dim Up", colour toggle: P_Rum_5_356.arrfbLysGruppe[1].fbLightCtrl.bDimUp
    Rectangle (127,252 71x22), "Dim Dwn", colour toggle: P_Rum_5_356.arrfbLysGruppe[1].fbLightCtrl.bDimDwn
    Ellipse (45,219 22x23), colour toggle: P_Rum_5_356.arrfbLysGruppe[1].fbLightCtrl.bAutoZone1
    Rectangle (78,219 122x22), "Lys Auto"
    Ellipse (45,54 22x23), colour toggle: P_Gang_5_356.arrfbLysGruppe[1].fbLightCtrl.bPIR
    Rectangle (77,54 122x22), "PIR status"
END_VISUALIZATION

// ---- POUs/Alle_Rum/Rum_Med_DALI_Pir/Rum_4_407/Visualization_5_356_2_1_1_6_1_6_1.TcVIS
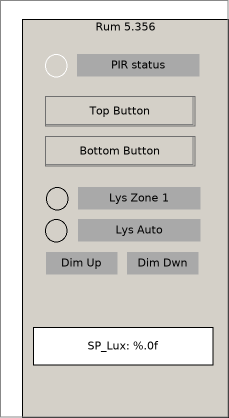
VISUALIZATION Visualization_5_356_2_1_1_6_1_6_1  // 229x418
    RoundedRectangle (22,19 207x399), "Rum 5.356"
    Rectangle (33,327 180x38), "SP_Lux: %.0f", text variable: P_Rum_5_356.arrfbLysGruppe[1].fbLightCtrl.fLuxZone1
    Button (45,96 150x30), "Top Button"
        tap P_Rum_5_356.bTopButtonZone1_Visu
    Button (45,136 150x30), "Bottom Button"
        tap P_Rum_5_356.bBottomButtonZone1_Visu
    Ellipse (46,187 22x23), colour toggle: P_Rum_5_356.arrfbLysGruppe[1].fbLightCtrl.bOnZone1
    Rectangle (78,187 122x22), "Lys Zone 1"
    Rectangle (46,252 71x22), "Dim Up", colour toggle: P_Rum_5_356.arrfbLysGruppe[1].fbLightCtrl.bDimUp
    Rectangle (127,252 71x22), "Dim Dwn", colour toggle: P_Rum_5_356.arrfbLysGruppe[1].fbLightCtrl.bDimDwn
    Ellipse (45,219 22x23), colour toggle: P_Rum_5_356.arrfbLysGruppe[1].fbLightCtrl.bAutoZone1
    Rectangle (78,219 122x22), "Lys Auto"
    Ellipse (45,54 22x23), colour toggle: P_Gang_5_356.arrfbLysGruppe[1].fbLightCtrl.bPIR
    Rectangle (77,54 122x22), "PIR status"
END_VISUALIZATION

// ---- POUs/Alle_Rum/Rum_Med_DALI_Pir/Rum_3_429/Visualization_5_356_2_1_1_1_1_1.TcVIS
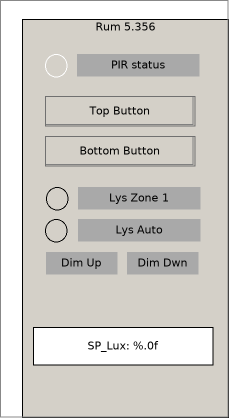
VISUALIZATION Visualization_5_356_2_1_1_1_1_1  // 229x418
    RoundedRectangle (22,19 207x399), "Rum 5.356"
    Rectangle (33,327 180x38), "SP_Lux: %.0f", text variable: P_Rum_5_356.arrfbLysGruppe[1].fbLightCtrl.fLuxZone1
    Button (45,96 150x30), "Top Button"
        tap P_Rum_5_356.bTopButtonZone1_Visu
    Button (45,136 150x30), "Bottom Button"
        tap P_Rum_5_356.bBottomButtonZone1_Visu
    Ellipse (46,187 22x23), colour toggle: P_Rum_5_356.arrfbLysGruppe[1].fbLightCtrl.bOnZone1
    Rectangle (78,187 122x22), "Lys Zone 1"
    Rectangle (46,252 71x22), "Dim Up", colour toggle: P_Rum_5_356.arrfbLysGruppe[1].fbLightCtrl.bDimUp
    Rectangle (127,252 71x22), "Dim Dwn", colour toggle: P_Rum_5_356.arrfbLysGruppe[1].fbLightCtrl.bDimDwn
    Ellipse (45,219 22x23), colour toggle: P_Rum_5_356.arrfbLysGruppe[1].fbLightCtrl.bAutoZone1
    Rectangle (78,219 122x22), "Lys Auto"
    Ellipse (45,54 22x23), colour toggle: P_Gang_5_356.arrfbLysGruppe[1].fbLightCtrl.bPIR
    Rectangle (77,54 122x22), "PIR status"
END_VISUALIZATION

// ---- POUs/DALI/DALI_Setup/VISUs/Visu_DALICommissioning/Visu_Part202Status.TcVIS
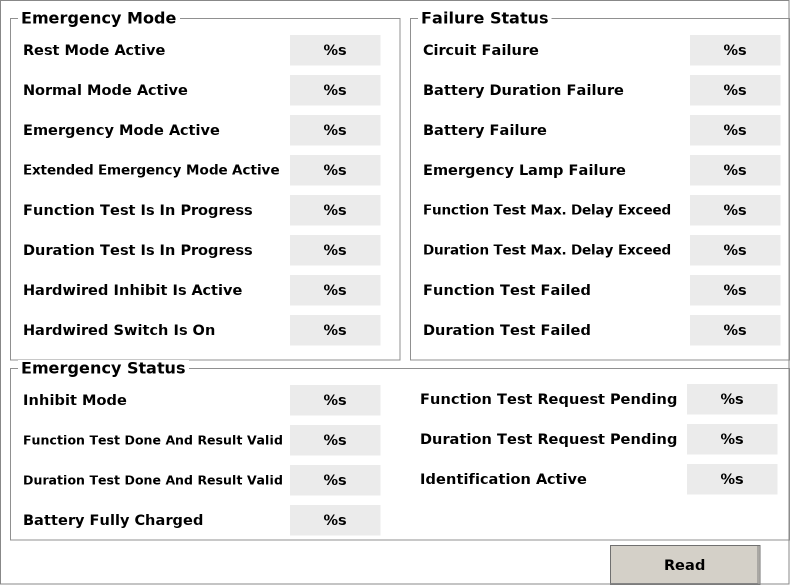
VISUALIZATION Visu_Part202Status  // 790x585
    Button (610,545 150x40), "Read"
        OnMouseClick: execute { DALI_Commissioning.fbPart202Emergency.bReadState:=TRUE; }
    GroupBox (10,10 390x350), "Emergency Mode"
        Textfield (10,145 260x30), "Extended Emergency Mode Active"
        Textfield (280,185 90x30), "%s", text variable: DALI_Commissioning.fbPart202Emergency.sFunctionTest
        Textfield (280,145 90x30), "%s", text variable: DALI_Commissioning.fbPart202Emergency.sExtendedEmergency
        Textfield (280,105 90x30), "%s", text variable: DALI_Commissioning.fbPart202Emergency.sEmergencyMode
        Textfield (280,65 90x30), "%s", text variable: DALI_Commissioning.fbPart202Emergency.sNormalMode
        Textfield (280,25 90x30), "%s", text variable: DALI_Commissioning.fbPart202Emergency.sRestMode
        Textfield (10,25 260x30), "Rest Mode Active"
        Textfield (10,65 260x30), "Normal Mode Active"
        Textfield (10,105 260x30), "Emergency Mode Active"
        Textfield (10,185 260x30), "Function Test Is In Progress"
        Textfield (10,225 260x30), "Duration Test Is In Progress"
        Textfield (10,265 260x30), "Hardwired Inhibit Is Active"
        Textfield (10,305 260x30), "Hardwired Switch Is On"
        Textfield (280,265 90x30), "%s", text variable: DALI_Commissioning.fbPart202Emergency.sHardwiredInhibit
        Textfield (280,305 90x30), "%s", text variable: DALI_Commissioning.fbPart202Emergency.sHardwiredSwitch
        Textfield (280,225 90x30), "%s", text variable: DALI_Commissioning.fbPart202Emergency.sDurationTest
    GroupBox (410,10 380x350), "Failure Status"
        Textfield (10,145 260x30), "Emergency Lamp Failure"
        Textfield (280,185 90x30), "%s", text variable: DALI_Commissioning.fbPart202Emergency.sFunctionTestExceed
        Textfield (280,145 90x30), "%s", text variable: DALI_Commissioning.fbPart202Emergency.sEmergencyLampFailure
        Textfield (280,105 90x30), "%s", text variable: DALI_Commissioning.fbPart202Emergency.sBatteryFailure
        Textfield (280,65 90x30), "%s", text variable: DALI_Commissioning.fbPart202Emergency.sBatteryDurationFailure
        Textfield (280,25 90x30), "%s", text variable: DALI_Commissioning.fbPart202Emergency.sCircuitFailure
        Textfield (10,25 260x30), "Circuit Failure"
        Textfield (10,65 260x30), "Battery Duration Failure"
        Textfield (10,105 260x30), "Battery Failure"
        Textfield (10,185 260x30), "Function Test Max. Delay Exceed"
        Textfield (10,225 260x30), "Duration Test Max. Delay Exceed"
        Textfield (10,265 260x30), "Function Test Failed"
        Textfield (10,305 260x30), "Duration Test Failed"
        Textfield (280,265 90x30), "%s", text variable: DALI_Commissioning.fbPart202Emergency.sFunctionTestFailed
        Textfield (280,305 90x30), "%s", text variable: DALI_Commissioning.fbPart202Emergency.sDurationTestFailed
        Textfield (280,225 90x30), "%s", text variable: DALI_Commissioning.fbPart202Emergency.sDurationTestExceed
    GroupBox (10,360 780x180), "Emergency Status"
        Textfield (10,145 260x30), "Battery Fully Charged"
        Textfield (677,24 90x30), "%s", text variable: DALI_Commissioning.fbPart202Emergency.sFunctionTestRequestPending
        Textfield (10,25 260x30), "Inhibit Mode"
        Textfield (10,65 260x30), "Function Test Done And Result Valid"
        Textfield (407,24 260x30), "Function Test Request Pending"
        Textfield (407,64 260x30), "Duration Test Request Pending"
        Textfield (407,104 260x30), "Identification Active"
        Textfield (677,104 90x30), "%s", text variable: DALI_Commissioning.fbPart202Emergency.sIdentificationActive
        Textfield (677,64 90x30), "%s", text variable: DALI_Commissioning.fbPart202Emergency.sDurationTestRequestPending
        Textfield (280,25 90x30), "%s", text variable: DALI_Commissioning.fbPart202Emergency.sInhibitMode
        Textfield (280,65 90x30), "%s", text variable: DALI_Commissioning.fbPart202Emergency.sFunctionTestDoneValid
        Textfield (280,145 90x30), "%s", text variable: DALI_Commissioning.fbPart202Emergency.sBatteryFullCharged
        Textfield (10,105 260x30), "Duration Test Done And Result Valid"
        Textfield (280,105 90x30), "%s", text variable: DALI_Commissioning.fbPart202Emergency.sDurationTestDoneValid
END_VISUALIZATION

// ---- POUs/DALI/DALI_Setup/VISUs/Visu_DALICommissioning/Visu_Part205.TcVIS
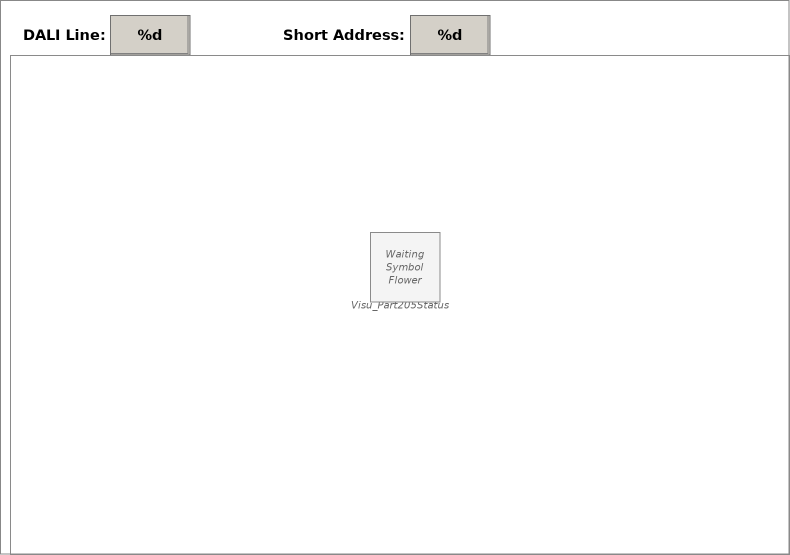
VISUALIZATION Visu_Part205  // 790x555
    Group (280,15 210x40)
        Textfield (0,0 130x40), "Short Address:"
        Button (130,0 80x40), "%d", text variable: DALI_Commissioning.fbPart205Incandescent.nAddress
            OnMouseClick: write the text variable via Default, min 0, max 63, title "Insert Short Address"
    Group (20,15 170x40)
        Textfield (0,0 110x40), "DALI Line:"
        Button (90,0 80x40), "%d", text variable: GVL_Internal.nDALILine
            OnMouseClick: write the text variable via Default, min 1, max 10, title "Choose line"
    TabControl (10,55 780x500)
        shows Visu_Part205Status()
        shows Visu_Part205Parameters()
        shows Visu_Part202Parameters()
        [0]: TabTitle=Status
        [1]: TabTitle=Parameters
        [2]: TabTitle=Parameters
    WaitingSymbolFlower (370,232 70x70), invisible if: DALI_Commissioning.fbPart205Incandescent.bHideWaitSymbol
END_VISUALIZATION

// ---- POUs/DALI/DALI_Setup/VISUs/Visu_DALICommissioning/Visu_Part205Parameters.TcVIS
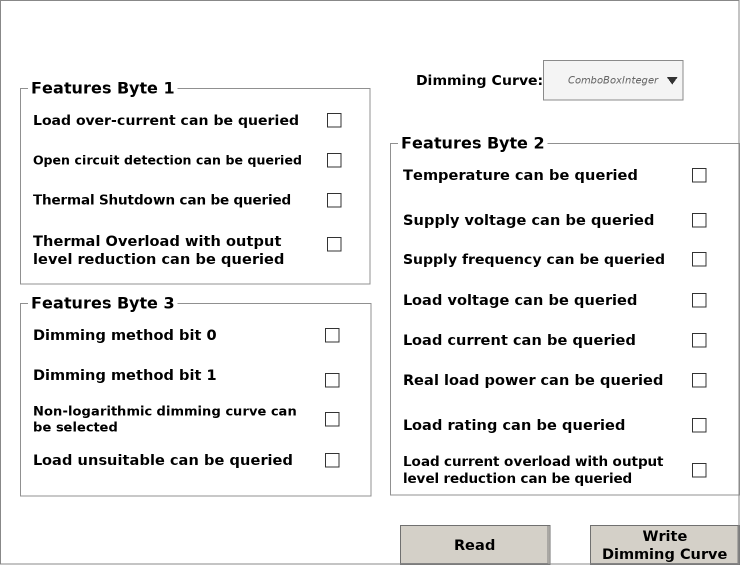
VISUALIZATION Visu_Part205Parameters  // 740x565
    Button (590,525 150x40), "Write Dimming Curve"
        OnMouseClick: execute { DALI_Commissioning.fbPart205Incandescent.bWrite := TRUE; }
    Button (400,525 150x40), "Read"
        OnMouseClick: execute { DALI_Commissioning.fbPart205Incandescent.bReadParameter := TRUE; }
    Group (413,60 270x40)
        Textfield (0,0 130x40), "Dimming Curve:"
        ComboBoxInteger (130,0 140x40), variable: DALI_Commissioning.fbPart205Incandescent.eDimmingCurve, text list: 'DimmingCurve'
    GroupBox (20,80 350x204), "Features Byte 1"
        Textfield (10,25 270x30), "Load over-current can be queried"
        Checkbox (305,25 30x30), variable: DALI_Commissioning.fbPart205Incandescent.bLoadOverCurrentShutdownQueried, input disabled if: True
        Textfield (10,65 270x30), "Open circuit detection can be queried"
        Textfield (10,105 270x30), "Thermal Shutdown can be queried"
        Checkbox (305,65 30x30), variable: DALI_Commissioning.fbPart205Incandescent.bOpenCircuitQueried, input disabled if: true
        Checkbox (305,105 30x30), variable: DALI_Commissioning.fbPart205Incandescent.bThermalShutdownQueried, input disabled if: True
        Textfield (10,150 270x40), "Thermal Overload with output level reduction can be queried"
    GroupBox (390,135 350x360), "Features Byte 2"
        Textfield (10,25 270x30), "Temperature can be queried"
        Checkbox (300,25 30x30), variable: DALI_Commissioning.fbPart205Incandescent.bTempQueried, input disabled if: True
        Textfield (10,65 270x30)
        Textfield (10,65 270x40), "Supply voltage can be queried"
        Textfield (10,150 270x30), "Load voltage can be queried"
        Textfield (10,109 270x30), "Supply frequency can be queried"
        Checkbox (300,70 30x30), variable: DALI_Commissioning.fbPart205Incandescent.bSupplyVoltageQueried, input disabled if: True
        Checkbox (300,150 30x30), variable: DALI_Commissioning.fbPart205Incandescent.bLoadVoltageQueried, input disabled if: True
        Checkbox (300,109 30x30), variable: DALI_Commissioning.fbPart205Incandescent.bSupplyFrequencyQueried, input disabled if: True
        Textfield (10,190 270x30), "Load current can be queried"
        Checkbox (300,190 30x30), variable: DALI_Commissioning.fbPart205Incandescent.bLoadCurrentQueried, input disabled if: True
        Textfield (10,230 270x30), "Real load power can be queried"
        Textfield (10,270 270x40), "Load rating can be queried"
        Textfield (10,320 270x30), "Load current overload with output level reduction can be queried"
        Checkbox (300,230 30x30), variable: DALI_Commissioning.fbPart205Incandescent.bRealLoadPowerQueried, input disabled if: True
        Checkbox (300,275 30x30), variable: DALI_Commissioning.fbPart205Incandescent.bLoadRatingQueried, input disabled if: True
        Checkbox (300,320 30x30), variable: DALI_Commissioning.fbPart205Incandescent.bLoadCurrentOverloadQueried
    GroupBox (20,295 351x201), "Features Byte 3"
        Textfield (10,25 270x30), "Dimming method bit 0"
        Checkbox (303,25 30x30), variable: DALI_Commissioning.fbPart205Incandescent.bDimmingMethodBit0, input disabled if: True
        Textfield (10,65 270x30)
        Textfield (10,65 270x30), "Dimming method bit 1"
        Textfield (10,150 270x30), "Load unsuitable can be queried"
        Textfield (10,109 270x30), "Non-logarithmic dimming curve can be selected"
        Checkbox (303,70 30x30), variable: DALI_Commissioning.fbPart205Incandescent.bDimmingMethodBit1, input disabled if: True
        Checkbox (303,150 30x30), variable: DALI_Commissioning.fbPart205Incandescent.bUnsuitableLoadQueried, input disabled if: True
        Checkbox (303,109 30x30), variable: DALI_Commissioning.fbPart205Incandescent.bNonLogarithmicCurve, input disabled if: True
    Checkbox (325,229 30x30), variable: DALI_Commissioning.fbPart205Incandescent.bThermalOverloadQueried, input disabled if: True
END_VISUALIZATION

// ---- POUs/DALI/DALI_Setup/VISUs/Visu_DALICommissioning/Visu_Part302AbsoluteInputDevice.TcVIS
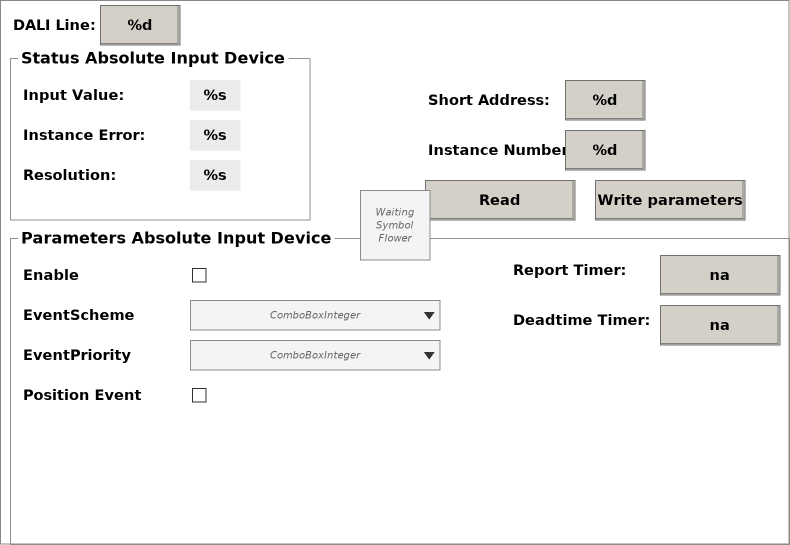
VISUALIZATION Visu_Part302AbsoluteInputDevice  // 790x545
    GroupBox (10,50 300x170), "Status Absolute Input Device"
        Textfield (10,30 160x30), "Input Value:"
        Textfield (10,70 160x30), "Instance Error:"
        Textfield (10,110 160x30), "Resolution:"
        Textfield (180,30 50x30), "%s", text variable: DALI_Commissioning.fbPart302AbsoluteInputDevice.nInputValue
        Textfield (180,70 50x30), "%s", text variable: DALI_Commissioning.fbPart302AbsoluteInputDevice.nInstanceError
        Textfield (180,110 50x30), "%s", text variable: DALI_Commissioning.fbPart302AbsoluteInputDevice.nResolution
    Button (425,180 150x40), "Read"
        OnMouseClick: execute { DALI_Commissioning.fbPart302AbsoluteInputDevice.bRead := TRUE; }
    GroupBox (10,230 780x315), "Parameters Absolute Input Device"
        Textfield (500,75 145x30), "Deadtime Timer:"
        Textfield (500,25 145x30), "Report Timer:"
        Textfield (10,30 150x30), "Enable"
        Button (650,25 120x40), "%d s", text variable: DALI_Commissioning.fbPart302AbsoluteInputDevice.nReport
            OnMouseClick: write DALI_Commissioning.fbPart302AbsoluteInputDevice.nReport via Default, min 0, max 255, title "Insert value for report timer"
        Button (650,75 120x40), "%d ms", text variable: DALI_Commissioning.fbPart302AbsoluteInputDevice.nDeadtime
            OnMouseClick: write DALI_Commissioning.fbPart302AbsoluteInputDevice.nDeadtime via Default, min 0, max 12750, title "Insert value for deadtime timer"
        Checkbox (180,30 30x30), variable: DALI_Commissioning.fbPart302AbsoluteInputDevice.bEnable
        Textfield (10,70 150x30), "EventScheme"
        ComboBoxInteger (180,70 250x30), variable: DALI_Commissioning.fbPart302AbsoluteInputDevice.eEventScheme, text list: 'EventScheme'
        Button (650,25 120x40), "na", invisible if: Not DALI_Commissioning.fbPart302AbsoluteInputDevice.bNoReportTimer, input disabled if: Not DALI_Commissioning.fbPart302AbsoluteInputDevice.bNoReportTimer
        Button (650,75 120x40), "na", invisible if: Not DALI_Commissioning.fbPart302AbsoluteInputDevice.bNoDeadtimeTimer, input disabled if: Not DALI_Commissioning.fbPart302AbsoluteInputDevice.bNoDeadtimeTimer
        Textfield (10,110 150x30), "EventPriority"
        Textfield (10,150 150x30), "Position Event"
        ComboBoxInteger (180,110 250x30), variable: DALI_Commissioning.fbPart302AbsoluteInputDevice.eEventPriority, text list: 'EventPriority'
        Checkbox (180,150 30x30), variable: DALI_Commissioning.fbPart302AbsoluteInputDevice.bPositionEventEnabled
    WaitingSymbolFlower (360,190 70x70), invisible if: DALI_Commissioning.fbPart302AbsoluteInputDevice.bHideWaitSymbol
    Button (595,180 150x40), "Write parameters"
        OnMouseClick: execute { DALI_Commissioning.fbPart302AbsoluteInputDevice.bWrite := TRUE; }
    Group (10,5 170x40)
        Textfield (0,0 110x40), "DALI Line:"
        Button (90,0 80x40), "%d", text variable: GVL_Internal.nDALILine
            OnMouseClick: write the text variable via Default, min 1, max 10, title "Choose line"
    Textfield (425,80 130x40), "Short Address:"
    Button (565,80 80x40), "%d", text variable: DALI_Commissioning.fbPart302AbsoluteInputDevice.nAddress
        OnMouseClick: write DALI_Commissioning.fbPart302AbsoluteInputDevice.nAddress via Default, min 0, max 63, title "Insert Short Address"
    Textfield (425,130 150x40), "Instance Number:"
    Button (565,130 80x40), "%d", text variable: DALI_Commissioning.fbPart302AbsoluteInputDevice.nInstanceAddress
        OnMouseClick: write DALI_Commissioning.fbPart302AbsoluteInputDevice.nInstanceAddress via Default, min 0, max 31, title "Insert instance number"
END_VISUALIZATION
